# EPICS substitutions: pvScanApp/Db/pv.substitutions
file pvCommon.template {
pattern
{none}
{none}
}

file scanPv.template {
pattern
{N, PREC}
{ 1,   3}
{ 2,   3}
{ 3,   3}
{ 4,   3}
{ 5,   3}
{ 6,   3}
{ 7,   3}
{ 8,   3}
{ 9,   3}
{10,   3}
}

file shutter.template {
pattern
{ N}
{ 1}
{ 2}
{ 3}
{ 4}
{ 5}
}
